PROGRAM MAIN
VAR
	input : ARRAY[0..4] OF LREAL := [1,1,1,1,1];
	out : ARRAY[0..0] OF LREAL;
	FB_nn : FB_Dense_v1;
END_VAR

FB_nn(pointer_input := ADR(input),pointer_output:=ADR(out));

END_PROGRAM

(* stored: Version 1.1.0.1, ProductVersion 3.1.4024.12
   POU MAIN: Id {06a88f9f-d222-4935-a655-040178e44248}, SpecialFunc None *)
